FUNCTION_BLOCK AD_LAST_2 (* MERGE 2 AD in 1 AD (LAST WRITER WINS, nicht naiv gemergt) - welcher der beiden Sockets zuletzt geschrieben hat, gewinnt und wird sofort an OUT durchgereicht *)
  (* Standard: 61499-2; Description: Copyright (c) 2026 Meisterschulen am Ostbahnhof This program and the accompanying materials are made available under the terms of the Eclipse Public License 2.0 which is available at https://www.eclipse.org/legal/epl-2.0/ SPDX-License-Identifier: EPL-2.0 *)
  (* Version 1.0, 2026-08-31, Franz Höpfinger, Meisterschulen am Ostbahnhof, generic 2-way AD last-writer-wins merge, plain BasicFB (like E_D_FF/E_SR) instead of wiring F_SEL/E_RS inline every time - whichever Socket's own event fires IS the last-writer signal, no SR-latch needed *)
  PACKAGE adapter::events::unidirectional;
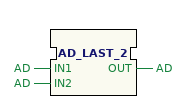
  SOCKETS
    IN1 : adapter::types::unidirectional::AD;
    IN2 : adapter::types::unidirectional::AD;
  END_SOCKETS
  PLUGS
    OUT : adapter::types::unidirectional::AD;
  END_PLUGS
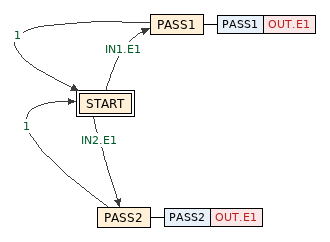
  EC_STATES
    START; (* Initial State *)
    PASS1 : PASS1 -> OUT.E1; (* IN1 zuletzt geschrieben *)
    PASS2 : PASS2 -> OUT.E1; (* IN2 zuletzt geschrieben *)
  END_STATES
  EC_TRANSITIONS
    START TO PASS1 := IN1.E1;
    START TO PASS2 := IN2.E1;
    PASS2 TO START := 1;
    PASS1 TO START := 1;
  END_TRANSITIONS
  ALGORITHM PASS1 IN ST: (* IN1 durchreichen *)
OUT.D1 := IN1.D1;
  END_ALGORITHM
  ALGORITHM PASS2 IN ST: (* IN2 durchreichen *)
OUT.D1 := IN2.D1;
  END_ALGORITHM
END_FUNCTION_BLOCK
